INTERFACE I_SafetyProvider

PROPERTY P_EStopOK : BOOL
GET
END_GET
END_PROPERTY

PROPERTY P_ReadFromSafetyController : BOOL
GET
END_GET
END_PROPERTY

PROPERTY P_STO_OK : BOOL
GET
END_GET
END_PROPERTY

END_INTERFACE

(* stored: Version 1.1.0.1
   Itf I_SafetyProvider: Id {4f0b34bb-be6f-0ca8-1703-e0e6a327c684}
   Property P_EStopOK: Id {393f352d-ddaa-041e-3f1e-09c38a700023}
   Get Get: Id {f3bb6b2f-7774-0bcf-2603-feb48c686c2b}
   Property P_ReadFromSafetyController: Id {37429123-dfc8-094c-14f3-b409e7f1bd57}
   Get Get: Id {9acdedb9-cc80-0d91-22d1-433682fabb15}
   Property P_STO_OK: Id {669ce2fb-649b-0caa-1072-9c3e66e1b90d}
   Get Get: Id {676a6f88-04bc-0d3e-1fd5-3e92ef4f55d0} *)
